TYPE DUT_RECIPEOFFER :
STRUCT
	Dummy:			BOOL := TRUE;
	Name:			STRING[255]:= 'e.g. Product x';
	RecipeID:		INT;
	Description:	STRING[80]:= '%Description of the Recipe e.g. "a recipe, that produces a product with feature x"';
	UserParameter:  ARRAY [0..UserParameterCnt] OF DUT_RECIPE_USERPARAMETEROUTPUT;
END_STRUCT
END_TYPE

(* stored: Version 1.1.0.1, ProductVersion 3.1.0.25
   DUT DUT_RECIPEOFFER: Id {bd3034e5-3021-47c6-9db0-d2025ca7a676} *)
